// LS Electric XG5000 project: 사칙연산
// PLC LSPLC
// module base 0 slot 0: 입출력 모듈:XBC-DR14E (DC 24V 입력 8점, 릴레이 출력 6점)

PROGRAM NewProgram (task: 스캔 프로그램)

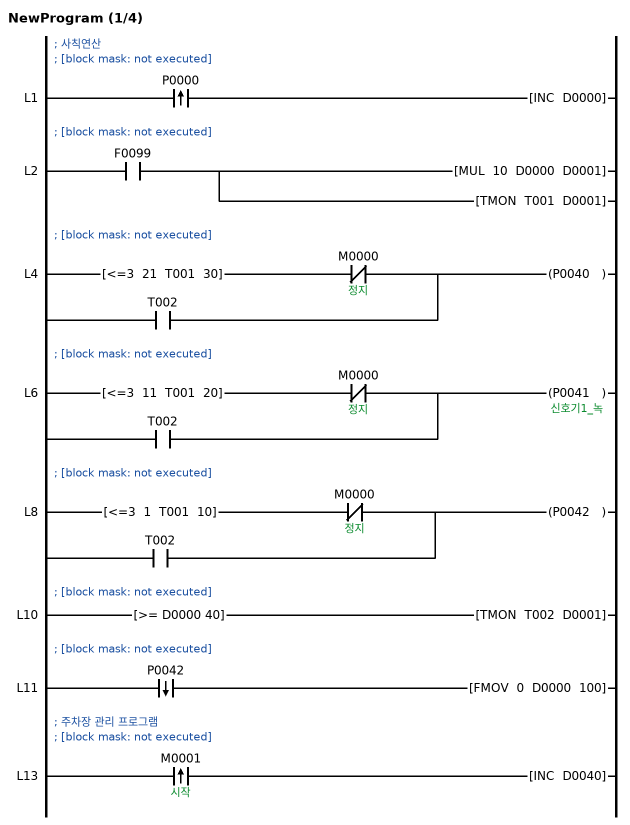
// 사칙연산
; L1 (block mask: not executed)
LOADP     P0000
INC       D0000
; L2 (block mask: not executed)
LOAD      F0099
MUL       10 D0000 D0001
TMON      T001 D0001
; L4 (block mask: not executed)
LOAD<=3   21 T001 30
AND NOT   M0000	// 정지
OR        T002
OUT       P0040
; L6 (block mask: not executed)
LOAD<=3   11 T001 20
AND NOT   M0000	// 정지
OR        T002
OUT       P0041	// 신호기1_녹
; L8 (block mask: not executed)
LOAD<=3   1 T001 10
AND NOT   M0000	// 정지
OR        T002
OUT       P0042
; L10 (block mask: not executed)
LOAD>=    D0000 40
TMON      T002 D0001
; L11 (block mask: not executed)
LOADN     P0042
FMOV      0 D0000 100
// 주차장 관리 프로그램
; L13 (block mask: not executed)
LOADP     M0001	// 시작
INC       D0040

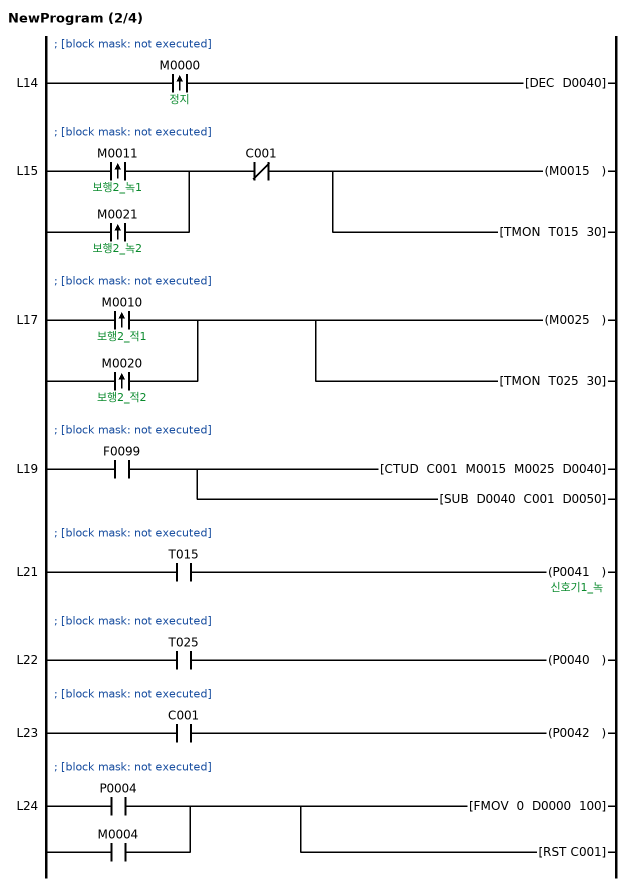
; L14 (block mask: not executed)
LOADP     M0000	// 정지
DEC       D0040
; L15 (block mask: not executed)
LOADP     M0011	// 보행2_녹1
ORP       M0021	// 보행2_녹2
AND NOT   C001
OUT       M0015
TMON      T015 30
; L17 (block mask: not executed)
LOADP     M0010	// 보행2_적1
ORP       M0020	// 보행2_적2
OUT       M0025
TMON      T025 30
; L19 (block mask: not executed)
LOAD      F0099
CTUD      C001 M0015 M0025 D0040
SUB       D0040 C001 D0050
; L21 (block mask: not executed)
LOAD      T015
OUT       P0041	// 신호기1_녹
; L22 (block mask: not executed)
LOAD      T025
OUT       P0040
; L23 (block mask: not executed)
LOAD      C001
OUT       P0042
; L24 (block mask: not executed)
LOAD      P0004
OR        M0004
FMOV      0 D0000 100
RST       C001

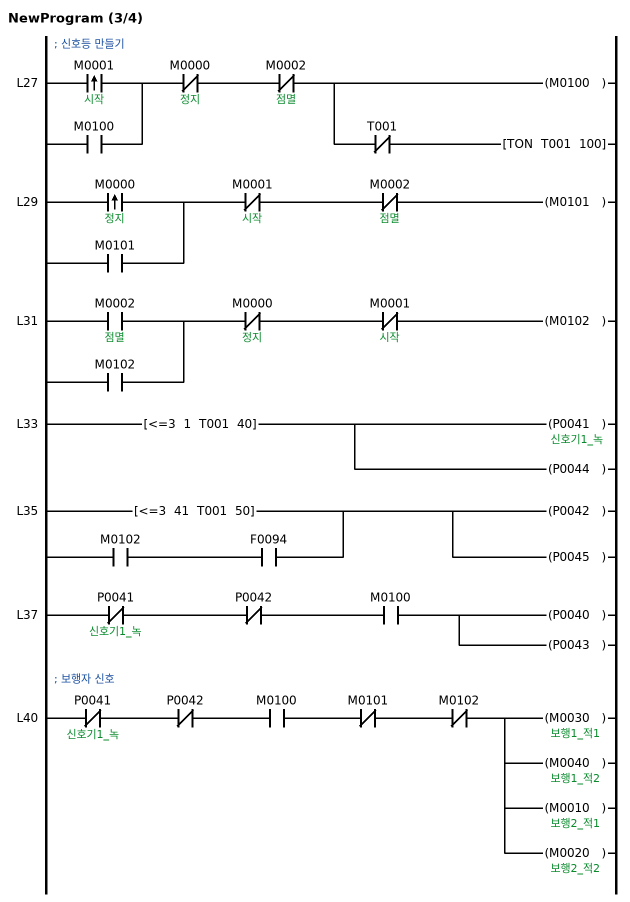
// 신호등 만들기
; L27
LOADP     M0001	// 시작
OR        M0100
AND NOT   M0000	// 정지
AND NOT   M0002	// 점멸
OUT       M0100
AND NOT   T001
TON       T001 100
; L29
LOADP     M0000	// 정지
OR        M0101
AND NOT   M0001	// 시작
AND NOT   M0002	// 점멸
OUT       M0101
; L31
LOAD      M0002	// 점멸
OR        M0102
AND NOT   M0000	// 정지
AND NOT   M0001	// 시작
OUT       M0102
; L33
LOAD<=3   1 T001 40
OUT       P0041	// 신호기1_녹
OUT       P0044
; L35
LOAD<=3   41 T001 50
LOAD      M0102
AND       F0094
OR LOAD
OUT       P0042
OUT       P0045
; L37
LOAD NOT  P0041	// 신호기1_녹
AND NOT   P0042
AND       M0100
OUT       P0040
OUT       P0043
// 보행자 신호
; L40
LOAD NOT  P0041	// 신호기1_녹
AND NOT   P0042
AND       M0100
AND NOT   M0101
AND NOT   M0102
OUT       M0030	// 보행1_적1
OUT       M0040	// 보행1_적2
OUT       M0010	// 보행2_적1
OUT       M0020	// 보행2_적2

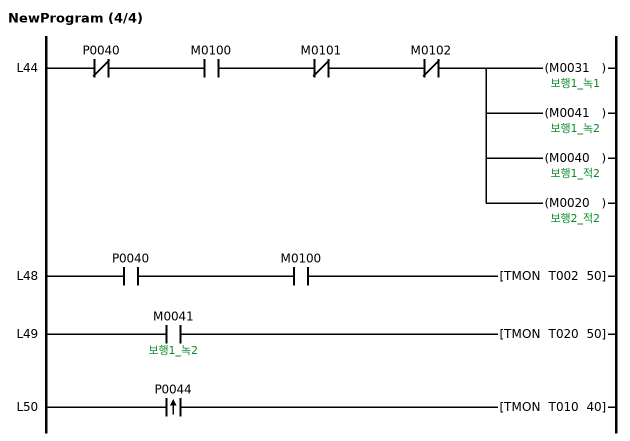
; L44
LOAD NOT  P0040
AND       M0100
AND NOT   M0101
AND NOT   M0102
OUT       M0031	// 보행1_녹1
OUT       M0041	// 보행1_녹2
OUT       M0040	// 보행1_적2
OUT       M0020	// 보행2_적2
; L48
LOAD      P0040
AND       M0100
TMON      T002 50
; L49
LOAD      M0041	// 보행1_녹2
TMON      T020 50
; L50
LOADP     P0044
TMON      T010 40